FUNCTION_BLOCK FB_SelectOperatorExample

VAR
	test1, result1, result2, lowerLimit, upperLimit : DINT;
	test2 : BOOL;
END_VAR

result1 := LIMIT(lowerLimit, test1 ,upperLimit);

result2 := SEL(test2, 1, 2);

END_FUNCTION_BLOCK

(* stored: Version 1.1.0.1
   POU FB_SelectOperatorExample: Id {bca8ed81-aed1-4623-b87d-47a9bba08087}, SpecialFunc None *)
